FUNCTION_BLOCK FB_3HeaterControl
VAR_INPUT
	m_Enbale					: BOOL;
	m_Temperature_high			: BOOL;
	m_Battery_Discharging		: BOOL;
	real_Temperature			: REAL;
	real_TemperatureSetPoint	: REAL;
	real_GridPower				: REAL;
	real_BatteryPower			: REAL;
	real_Size_Step1_kW			: REAL;
	real_Size_Step2_kW			: REAL;
	real_Size_Step3_kW			: REAL;
	
	
END_VAR
VAR_OUTPUT
	m_Step1						: BOOL;
	m_Step2						: BOOL;
	m_Step3						: BOOL;
END_VAR
VAR
	fb_HourCounter_Step1		: FB_HourCounter;
	fb_HourCounter_Step2		: FB_HourCounter;
	fb_HourCounter_Step3		: FB_HourCounter;
	r_Trig_allOff				: r_trig;
	real_Hours_Step1			: REAL;
	real_Hours_Step2			: REAL;
	real_Hours_Step3			: REAL;	
	arr_sint_StartOrder			: ARRAY[1..3] OF SINT;
	arr_real_LoadSize			: ARRAY[1..3] OF REAL;
	arr_real_Steps				: ARRAY[1..3] OF REAL;
	
	
	int_state					: INT;
	ton_OnDelay_Steps			: Ton;
	time_OnDelay				: TIME:=T#30S;	
	ton_OffDelay_Steps			: Ton;
	time_OffDelay				: TIME:=T#30S;	
	ton_WaitDelay_Steps			: Ton;
	time_WaitDelay				: TIME:=T#30S;	
	sint_Steps_On				: SINT;
	ton_OffDelay2_Steps			: Ton;
	time_OffDelay2				: TIME:=T#15S;	
END_VAR


CASE int_state OF
	0:	// not enabled
		m_Step1 := FALSE;
		m_Step2 := FALSE;
		m_Step3 := FALSE;
		sint_Steps_On := 0;
		ton_OnDelay_Steps.IN := FALSE;
		ton_OffDelay_Steps.IN := FALSE;
		ton_OffDelay2_Steps.IN := FALSE;
		ton_WaitDelay_Steps.IN := FALSE;
		
		IF 	m_Enbale THEN
			int_state := 10;
		END_IF
	
	10: // check that mains power gets more negative thenn step power + 20%
		IF sint_Steps_On <3 THEN 
			IF real_GridPower + arr_real_LoadSize[sint_Steps_On+1]*1.2 < 0 AND NOT m_Temperature_high AND real_Temperature < (real_TemperatureSetPoint-2) THEN 
				ton_OnDelay_Steps.IN := TRUE;
			ELSE
				ton_OnDelay_Steps.IN := FALSE;
			END_IF
		END_IF
		IF ton_OnDelay_Steps.Q THEN
			ton_OnDelay_Steps.IN := FALSE;
			int_state := 11;
		END_IF
		IF sint_Steps_On <>0 THEN 
			IF real_GridPower > 3 OR  real_Temperature > real_TemperatureSetPoint OR (m_Battery_Discharging AND real_BatteryPower > 5) THEN
 				ton_OffDelay_Steps.IN := TRUE;
			ELSE
				ton_OffDelay_Steps.IN := FALSE;
			END_IF
			IF real_GridPower > 10 THEN
 				ton_OffDelay2_Steps.IN := TRUE;
			ELSE
				ton_OffDelay2_Steps.IN := FALSE;
			END_IF
			
			IF ton_OffDelay_Steps.Q THEN
				ton_OffDelay_Steps.IN := FALSE;
				ton_OffDelay2_Steps.IN := FALSE;
				int_state := 12;
			END_IF
			IF m_Temperature_high AND sint_Steps_On <>0 THEN
				ton_OnDelay_Steps.IN := FALSE;
 				ton_OffDelay_Steps.IN := FALSE;
				ton_OffDelay2_Steps.IN := FALSE;
				int_state := 15;
			END_IF
		END_IF
		
		
	11: // count step one up
		sint_Steps_On := sint_Steps_On+1;
		int_state := 20;
		
	12:// count step one down
		sint_Steps_On := sint_Steps_On-1;
		int_state := 20;
	
	15:// Switch off all steps
		sint_Steps_On := 0;
		int_state := 20;
	
	20: // wait state	
		ton_WaitDelay_Steps.IN := TRUE;
		IF ton_WaitDelay_Steps.Q THEN
			ton_WaitDelay_Steps.IN := FALSE;
			int_state := 10;
		END_IF
END_CASE
ton_OnDelay_Steps(PT := time_OnDelay);
ton_OffDelay_Steps(PT := time_OffDelay);
ton_OffDelay2_Steps(PT := time_OffDelay2);
ton_WaitDelay_Steps(PT := time_WaitDelay);

// if not enabled, force state to 0
IF 	NOT m_Enbale THEN
	int_state := 0;
END_IF

// switch on steps according to sint_Steps_On
CASE sint_Steps_On OF
	0:
		m_Step1 := FALSE;
		m_Step2 := FALSE;
		m_Step3 := FALSE;
		
	1:
		m_Step1 := FALSE;
		m_Step2 := FALSE;
		m_Step3 := FALSE;
		IF arr_sint_StartOrder[1] = 1 THEN 
 			m_Step1 := TRUE;
		ELSIF arr_sint_StartOrder[1] = 2 THEN 
			m_Step2 := TRUE;
		ELSIF arr_sint_StartOrder[1] = 3 THEN 
			m_Step3 := TRUE;
		END_IF
	2:
		m_Step1 := FALSE;
		m_Step2 := FALSE;
		m_Step3 := FALSE;
		IF arr_sint_StartOrder[1] = 1 THEN 
 			m_Step1 := TRUE;
		ELSIF arr_sint_StartOrder[1] = 2 THEN 
			m_Step2 := TRUE;
		ELSIF arr_sint_StartOrder[1] = 3 THEN 
			m_Step3 := TRUE;
		END_IF
		IF arr_sint_StartOrder[2] = 1 THEN 
 			m_Step1 := TRUE;
		ELSIF arr_sint_StartOrder[2] = 2 THEN 
			m_Step2 := TRUE;
		ELSIF arr_sint_StartOrder[2] = 3 THEN 
			m_Step3 := TRUE;
		END_IF
	3:
		m_Step1 := TRUE;
		m_Step2 := TRUE;
		m_Step3 := TRUE;		
END_CASE		
	
// find out which step has the lowest running hours
r_Trig_allOff(CLK := NOT m_Step1 AND NOT m_Step2 AND NOT m_Step3);

IF r_Trig_allOff.Q THEN
	IF real_Hours_Step1 <= real_Hours_Step2 AND real_Hours_Step1<=real_Hours_Step3 THEN
		arr_sint_StartOrder[1] := 1;
		IF real_Hours_Step2 <= real_Hours_Step3 THEN
			arr_sint_StartOrder[2] := 2;
			arr_sint_StartOrder[3] := 3;
		ELSE
			arr_sint_StartOrder[2] := 3;
			arr_sint_StartOrder[3] := 2;
		END_IF
	ELSIF real_Hours_Step2 <= real_Hours_Step1 AND real_Hours_Step2<=real_Hours_Step3 THEN
		arr_sint_StartOrder[1] := 2;
		IF real_Hours_Step1 <= real_Hours_Step3 THEN
			arr_sint_StartOrder[2] := 1;
			arr_sint_StartOrder[3] := 3;
		ELSE
			arr_sint_StartOrder[2] := 3;
			arr_sint_StartOrder[3] := 1;
		END_IF
	ELSIF real_Hours_Step3 <= real_Hours_Step1 AND real_Hours_Step3<=real_Hours_Step2 THEN
		arr_sint_StartOrder[1] := 3;
		IF real_Hours_Step1 <= real_Hours_Step2 THEN
			arr_sint_StartOrder[2] := 1;
			arr_sint_StartOrder[3] := 2;
		ELSE
			arr_sint_StartOrder[2] := 2;
			arr_sint_StartOrder[3] := 1;
		END_IF
	END_IF
	arr_real_Steps[1]	:= real_Size_Step1_kW;
	arr_real_Steps[2]	:= real_Size_Step2_kW;
	arr_real_Steps[3]	:= real_Size_Step3_kW;
	
	arr_real_LoadSize[1] :=   arr_real_Steps[arr_sint_StartOrder[1]];
	arr_real_LoadSize[2] :=   arr_real_Steps[arr_sint_StartOrder[2]];
	arr_real_LoadSize[3] :=   arr_real_Steps[arr_sint_StartOrder[3]];
	
END_IF



// hour counter for each step
fb_HourCounter_Step1(	mCounterON:= m_Step1, 
						realHours=> real_Hours_Step1);
						
fb_HourCounter_Step2(	mCounterON:= m_Step2, 
						realHours=> real_Hours_Step2);
						
fb_HourCounter_Step3(	mCounterON:= m_Step3, 
						realHours=> real_Hours_Step3);

END_FUNCTION_BLOCK

(* stored: Version 1.1.0.1, ProductVersion 3.1.4024.12
   POU FB_3HeaterControl: Id {e354d3ea-6faf-4aea-9d12-8fcd8611e5de}, SpecialFunc None *)
